FUNCTION_BLOCK VALUES2ARRAY_2_LREAL (* Service Interface Function Block Type *)
  PACKAGE eclipse4diac::convert;
  {SET_ATTRIBUTE(eclipse4diac::core::GenericClassName, 'GEN_VALUES2ARRAY')}
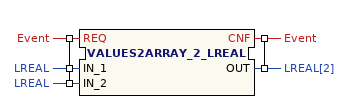
  EVENT_INPUT
    REQ WITH IN_1, IN_2; (* Service Request *)
  END_EVENT
  EVENT_OUTPUT
    CNF WITH OUT; (* Confirmation of Requested Service *)
  END_EVENT
  VAR_INPUT
    IN_1 : LREAL; (* input number 1 *)
    IN_2 : LREAL; (* input number 2 *)
  END_VAR
  VAR_OUTPUT
    OUT : ARRAY [0..1] OF LREAL; (* Array output *)
  END_VAR
END_FUNCTION_BLOCK
